FUNCTION_BLOCK SCALE_UR (* Scaling of a UINT input to a REAL range of{0.0..1.0} *)
  (* Standard: IEC 61499-1; Classification: Math; ApplicationDomain: Process Control, HVAC; Function: Scaling; Type: UINT to REAL; Description: Scaling a UINT to a REAL range of {0.0..1.0} *)
  (* Version 0.1, 2006-05-03, JHC, Holobloc Inc, Corrected documentation of OUT. *)
  (* Version 0.0, 2006-04-28, JHC, Holobloc Inc *)
  (* Compiler header: package fb.rt.hvac; *)
  (* Compiler Java Sun JDK 1.5.0 *)
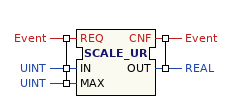
  EVENT_INPUT
    REQ WITH IN, MAX; (* Normal Execution Request *)
  END_EVENT
  EVENT_OUTPUT
    CNF WITH OUT; (* Execution Confirmation *)
  END_EVENT
  VAR_INPUT
    IN : UINT; (* Process (typically A/D) input *)
    MAX : UINT; (* IN value corrsponding to OUT=1.0 *)
  END_VAR
  VAR_OUTPUT
    OUT : REAL; (* Scaled Output, limited to {0.0..1.0} *)
  END_VAR
END_FUNCTION_BLOCK
